// TIA Portal V18 export
VAR_GLOBAL   // PLC tag table "11 Costanti Pressa"
END_VAR
VAR_GLOBAL CONSTANT   // user constants
   T50RCE : Int := 1;
   T400DM : Int := 9;
   T250DM : Int := 8;
   T200DM : Int := 7;
   T125DM : Int := 6;
   T100DM : Int := 5;
   T100RCE : Int := 4;
   T80RCE : Int := 3;
   T63RCE : Int := 2;
   T160DM : Int := 10;
END_VAR
